{attribute 'qualified_only'}
VAR_GLOBAL CONSTANT
	nMaxDebugArraySize		: UDINT := 10;
END_VAR

(* stored: Version 1.1.0.1
   GVL Param: Id {ccb9fd62-55b3-4cfe-888a-93eccd52e1bc}, ParameterList True *)
